FUNCTION TryConvert_ULINT_TO_UDINT : BOOL
VAR_INPUT
	in : ULINT;
	out : REFERENCE TO UDINT;
END_VAR

IF in > DatatypeLimits.MAX_VALUE_OF_ULINT_WHICH_CAN_BE_HELD_IN_A_UDINT THEN
	RETURN;
END_IF

out := ULINT_TO_UDINT(in);
TryConvert_ULINT_TO_UDINT := TRUE;

END_FUNCTION

(* stored: Version 1.1.0.1, ProductVersion 3.1.4024.12
   POU TryConvert_ULINT_TO_UDINT: Id {a7aaff76-d079-47a0-a391-726940de699c}, SpecialFunc None *)
